// TIA Portal V17 export
// export: Created 2023-02-26T22:28:44.481515Z, ExportSetting WithDefaults, DisplayName Totally Integrated Automation Portal, DisplayVersion V17, DisplayName TIA Portal Openness, DisplayVersion V17, DisplayName TIA Portal Version Control Interface, DisplayVersion V17, DisplayName TIA Portal Test Suite Advanced, DisplayVersion V17, DisplayName STEP 7 Professional, DisplayVersion V17, DisplayName SIMATIC Energy Suite, DisplayVersion V17, DisplayName STEP 7 Safety, DisplayVersion V17, DisplayName WinCC Professional, DisplayVersion V17
ORGANIZATION_BLOCK "Main"   // OB1, LAD, ProgramCycle
TITLE = "Main Program Sweep (Cycle)"
{ S7_Optimized_Access := 'TRUE' }
VERSION : 0.1
// stored: AutoNumber true, IsIECCheckEnabled false, SetENOAutomatically false
   VAR_INPUT
      Initial_Call : Bool;   // Initial call of this OB
      Remanence : Bool;   // =True, if remanent data are available
   END_VAR
BEGIN

REGION Network 1: Connection of PLC with FactoryIO
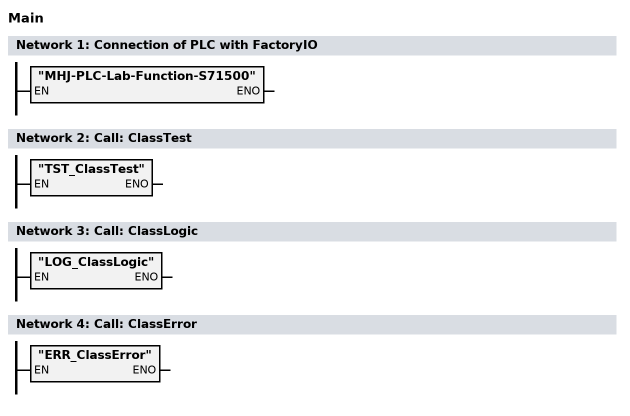
   RUNG wire#powerrail
      "MHJ-PLC-Lab-Function-S71500"()
   END_RUNG
   // the same network as SCL:
   "MHJ-PLC-Lab-Function-S71500"();
END_REGION

REGION Network 2: Call: ClassTest
   RUNG wire#powerrail
      "TST_ClassTest"()
   END_RUNG
   // the same network as SCL:
   "TST_ClassTest"();
END_REGION

REGION Network 3: Call: ClassLogic
   RUNG wire#powerrail
      "LOG_ClassLogic"()
   END_RUNG
   // the same network as SCL:
   "LOG_ClassLogic"();
END_REGION

REGION Network 4: Call: ClassError
   RUNG wire#powerrail
      "ERR_ClassError"()
   END_RUNG
   // the same network as SCL:
   "ERR_ClassError"();
END_REGION
END_ORGANIZATION_BLOCK
